KUKA KRL program: Looping.src

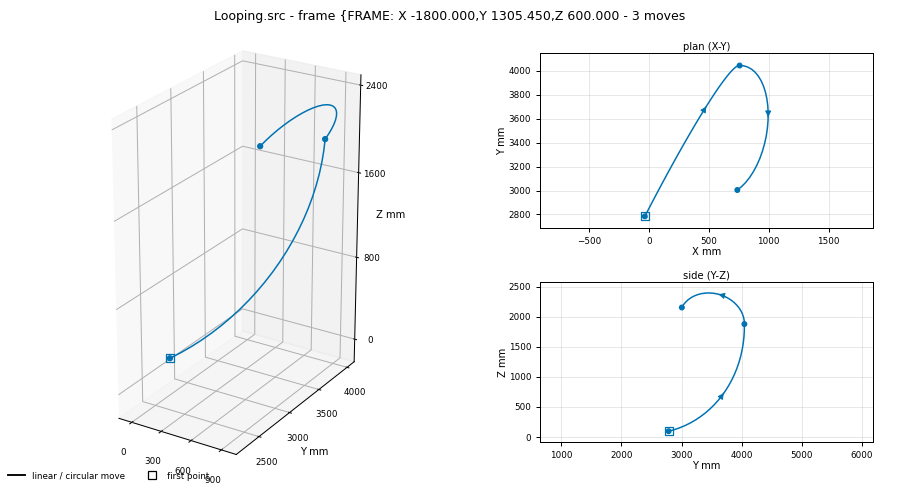
[picture p0: tool path of Looping.src in frame {FRAME: X -1800.000,Y 1305.450,Z 600.000, 3 of 5 moves have a stored position in this frame; points joined in program order, loops and branches not executed]
&ACCESS RVP
&REL 1
&PARAM TEMPLATE = C:\KRC\Roboter\Template\vorgabe
&PARAM EDITMASK = *
DEF Looping ( )
EXT BAS (BAS_COMMAND :IN,REAL :IN )


; GLOBAL INTERRUPT DECL 3 WHEN $STOPMESS==TRUE DO IR_STOPM ( )
; INTERRUPT ON 3

;FOLD Initialise and set default speed
BAS (#INITMOV,0)
BAS (#VEL_PTP,100)
BAS (#ACC_PTP,20)
$VEL.CP=0.2
BAS (#TOOL,0)
BAS (#BASE,0)
;ENDFOLD

;;FOLD STARTPOS
;$BWDSTART = FALSE
;PDAT_ACT = PDEFAULT
;BAS(#PTP_DAT)
;FDAT_ACT = {TOOL_NO 0,BASE_NO 0,IPO_FRAME #BASE}
;BAS(#FRAMES)
;;ENDFOLD

$ADVANCE = 5

;FOLD ---- Quickly skip BCO ----
; PTP $AXIS_ACT
;ENDFOLD

;FOLD ---- GO HOME ----
; PTP {A1 0.000, A2 -90.000, A3 90.000, A4 0.000, A5 0.000, A6 0.000, E1 0, E2 0, E3 0, E4 0, E5 0, E6 0}
;ENDFOLD


; Program generated by RoboDK v5.9.5 for KUKA KR 150 L120/2 on 12/01/2026 20:41:52
; Using nominal kinematics.
; ---- Setting reference (Base) ----
; BASE_DATA[2] = {FRAME: X -1800.000,Y 1305.450,Z 600.000,A -90.000,B 0.000,C 0.000}
$BASE = {FRAME: X -1800.000,Y 1305.450,Z 600.000,A -90.000,B 0.000,C 0.000}
; $BASE = BASE_DATA[2]
; --------------------------
; ---- Setting tool (TCP) ----
$TOOL = {FRAME: X 0.000,Y 0.000,Z 200.000,A 0.000,B 0.000,C 0.000}
; --------------------------
PTP {A1 -112.10300,A2 -65.54300,A3 134.78400,A4 -280.26200,A5 95.03930,A6 200.35700}
CIRC {X -82.589,Y 2226.590,Z -109.329,A 27.259,B 54.264,C -58.824},{X -35.213,Y 2784.400,Z 97.204,A 25.245,B 55.553,C -36.729}
CIRC {X 612.163,Y 3903.080,Z 1099.010,A 35.245,B 36.561,C -16.549},{X 756.652,Y 4044.400,Z 1878.600,A 13.630,B -14.594,C -6.382}
CIRC {X 995.043,Y 3609.130,Z 2375.820,A 18.407,B -45.817,C -8.879},{X 737.489,Y 3004.370,Z 2154.410,A -120.403,B -46.476,C 145.663}
PTP {A1 -49.74430,A2 -92.59980,A3 94.31610,A4 2.91424,A5 65.29800,A6 253.59600}
END
